FUNCTION_BLOCK earth_fault_5 (* Basic Function Block Type *)
  (* Standard: 61499-2 *)
  (* Version 0.0, 3/23/2016, gulzha, nxtControl GmbH, Template *)
  PACKAGE Main;
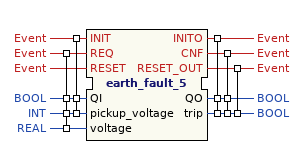
  EVENT_INPUT
    INIT WITH QI, pickup_voltage; (* Initialization Request *)
    REQ WITH QI, pickup_voltage, voltage; (* Normal Execution Request *)
    RESET;
  END_EVENT
  EVENT_OUTPUT
    INITO WITH QO, trip; (* Initialization Confirm *)
    CNF WITH QO, trip; (* Execution Confirmation *)
    RESET_OUT WITH trip;
  END_EVENT
  VAR_INPUT
    QI : BOOL; (* Input event qualifier *)
    pickup_voltage : INT;
    voltage : REAL;
  END_VAR
  VAR_OUTPUT
    QO : BOOL; (* Output event qualifier *)
    trip : BOOL;
  END_VAR
  VAR
    fault : BOOL;
    time2 : BOOL;
  END_VAR
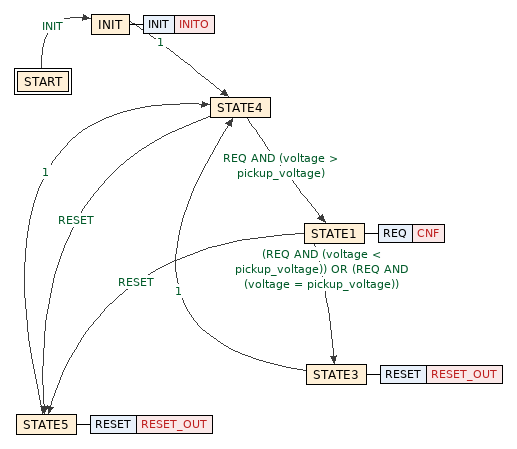
  EC_STATES
    START; (* Initial State *)
    INIT : INIT -> INITO; (* Initialization *)
    STATE1 : REQ -> CNF;
    STATE3 : RESET -> RESET_OUT;
    STATE5 : RESET -> RESET_OUT;
    STATE4;
  END_STATES
  EC_TRANSITIONS
    START TO INIT := INIT;
    INIT TO STATE4 := 1;
    STATE4 TO STATE1 := REQ AND (voltage > pickup_voltage);
    STATE1 TO STATE3 := (REQ AND (voltage < pickup_voltage)) OR (REQ AND (voltage = pickup_voltage));
    STATE5 TO STATE4 := 1;
    STATE4 TO STATE5 := RESET;
    STATE3 TO STATE4 := 1;
    STATE1 TO STATE5 := RESET;
  END_TRANSITIONS
  ALGORITHM INIT IN ST: (* Initialization algorithm *)
;

trip := FALSE;
fault := FALSE;
time2 := FALSE;
  END_ALGORITHM
  ALGORITHM REQ IN ST: (* Normally executed algorithm *)
;
trip := TRUE;
  END_ALGORITHM
  ALGORITHM RESET IN ST:
;

trip := FALSE;
fault := FALSE;
time2 := FALSE;
  END_ALGORITHM
  ALGORITHM REQ2 IN ST:
;
fault := TRUE;
  END_ALGORITHM
  ALGORITHM time2_up IN ST:
;
time2 := TRUE;
  END_ALGORITHM
END_FUNCTION_BLOCK
